// TIA Portal V19 export
TYPE "LEXCHANGETRAY_typeRollerIoSignalProcessValues"
// simulated: Bool
// trayAutomaticDischargeDetectionEm1: Bool
// trayAutomaticFeedingDetectionEm1: Bool
// restraintTrayAntiReverseDetection2Em1: Bool
// restraintTrayAntiReverseDetection1Em1: Bool
// stored: Access Published
   STRUCT
      simulated : Bool;
      trayAutomaticDischargeDetectionEm1 : Bool;
      trayAutomaticFeedingDetectionEm1 : Bool;
      restraintTrayAntiReverseDetection2Em1 : Bool;
      restraintTrayAntiReverseDetection1Em1 : Bool;
   END_STRUCT;
END_TYPE
